% RSLogix 500 project Vacuum Feedback Control without PID.RSS, saved by version 8.30.00.16 %
PROJECT "UNTITLED"    % processor: Bul.1763 MicroLogix 1100 Series B %

PROGRAM FILES
  LAD 2   4 rungs
  LAD 3 "IO"  3 rungs
  LAD 4 "CTRL"  11 rungs

DATA FILES
  O0 OUTPUT  4 elements
  I1 INPUT  6 elements
  S2 STATUS  66 elements
  B3 BINARY  1 elements
  T4 TIMER  1 elements
  C5 COUNTER  1 elements
  R6 CONTROL  1 elements
  N7 INTEGER  7 elements
  F8 FLOAT  4 elements

LADDER 2
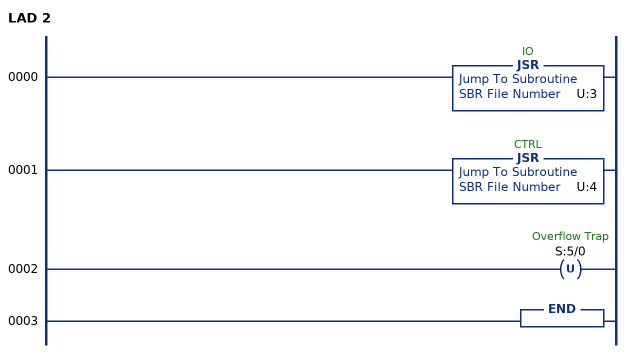
% Rung: 0 %
SOR JSR U:3 EOR
%   U:3  "IO" %
% Rung: 1 %
SOR JSR U:4 EOR
%   U:4  "CTRL" %
% Rung: 2 %
SOR OTU S:5/0 EOR
%   S:5/0  "Overflow Trap" %
% Rung: 3 %
SOR END EOR

LADDER 3 "IO"
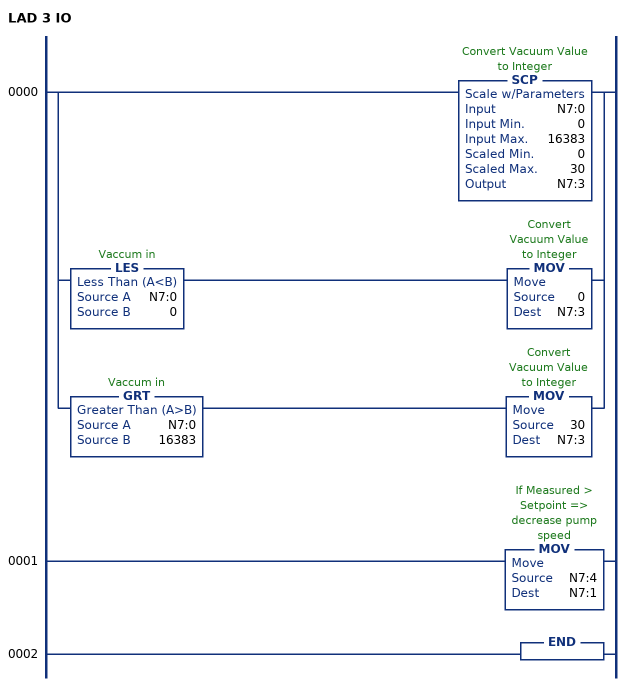
% Rung: 0 %
SOR BST SCP N7:0 0 16383 0 30 N7:3 NXB LES N7:0 0 MOV 0 N7:3 NXB GRT N7:0 16383 MOV 30 N7:3 BND EOR
%   N7:0  "Vaccum in" %
%   N7:3  "Convert Vacuum Value to Integer" %
% Rung: 1 %
SOR MOV N7:4 N7:1 EOR
%   N7:4  "(Measured - Setpoint)" %
%   N7:1  "If Measured > Setpoint => decrease pump speed" %
% Rung: 2 %
SOR END EOR

LADDER 4 "CTRL"
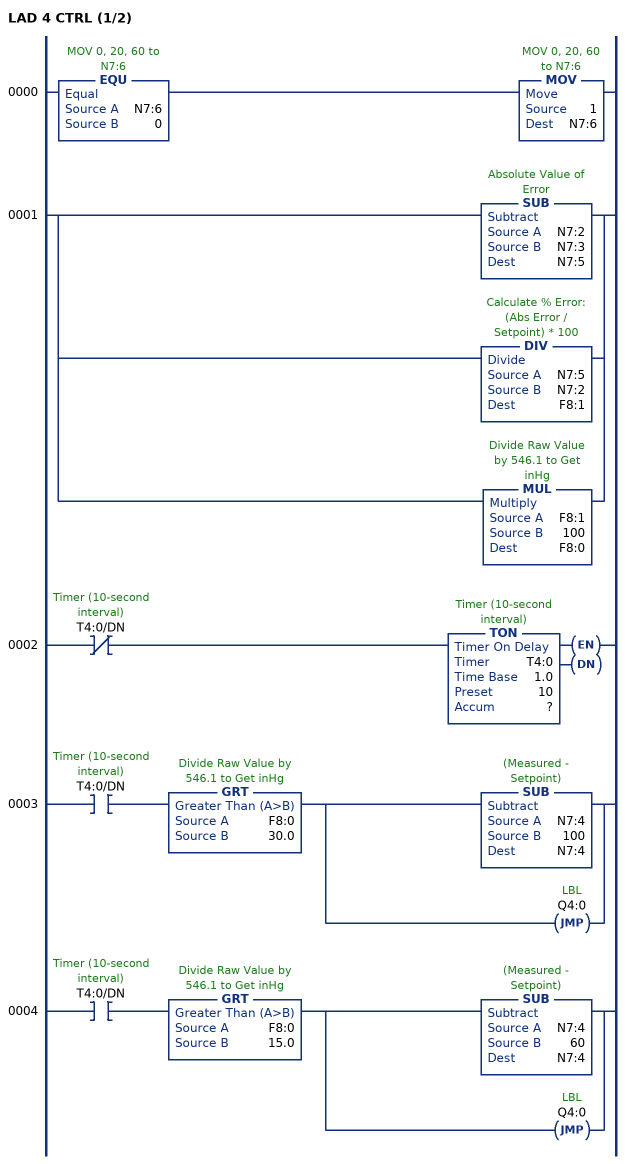
% Rung: 0 %
SOR EQU N7:6 0 MOV 1 N7:6 EOR
%   N7:6  "MOV 0, 20, 60 to N7:6" %
% Rung: 1 %
SOR BST SUB N7:2 N7:3 N7:5 NXB DIV N7:5 N7:2 F8:1 NXB MUL F8:1 100 F8:0 BND EOR
%   N7:2  "Calculate % Error: (Abs Error / Setpoint) * 100" %
%   N7:3  "Convert Vacuum Value to Integer" %
%   N7:5  "Absolute Value of Error" %
%   F8:1  "Calculate % Error: (Abs Error / Setpoint) * 100" %
%   F8:0  "Divide Raw Value by 546.1 to Get inHg" %
% Rung: 2 %  % edit flag set %
SOR XIO T4:0/DN TON T4:0 1.0 10 ? EOR
%   T4:0  "Timer (10-second interval)" %
% Rung: 3 %
SOR XIC T4:0/DN GRT F8:0 30.0 BST SUB N7:4 100 N7:4 NXB JMP Q4:0 BND EOR
%   T4:0  "Timer (10-second interval)" %
%   F8:0  "Divide Raw Value by 546.1 to Get inHg" %
%   N7:4  "(Measured - Setpoint)" %
%   Q4:0  "LBL" %
% Rung: 4 %
SOR XIC T4:0/DN GRT F8:0 15.0 BST SUB N7:4 60 N7:4 NXB JMP Q4:0 BND EOR
%   T4:0  "Timer (10-second interval)" %
%   F8:0  "Divide Raw Value by 546.1 to Get inHg" %
%   N7:4  "(Measured - Setpoint)" %
%   Q4:0  "LBL" %

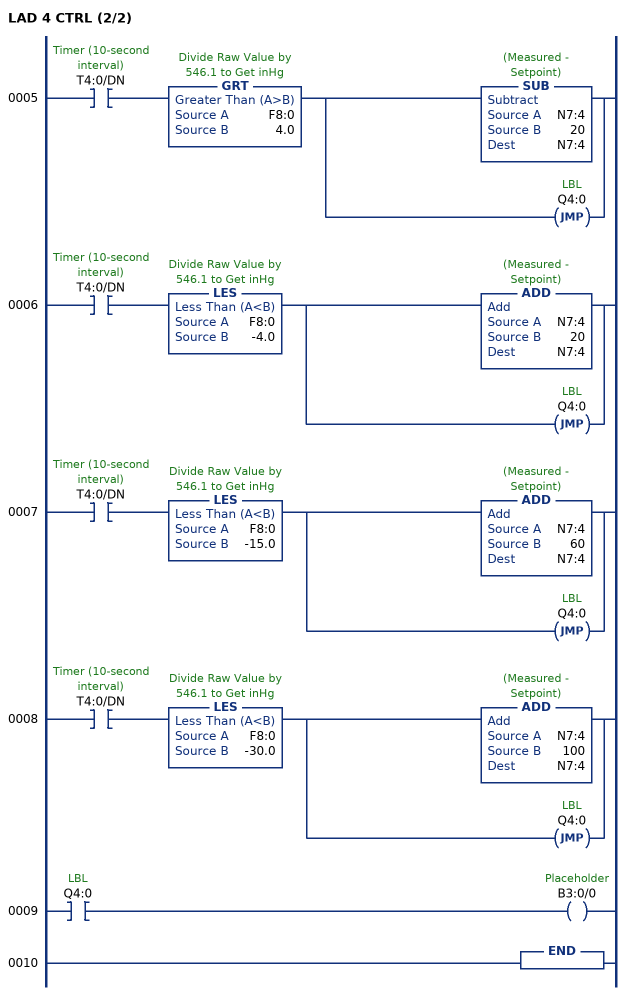
% Rung: 5 %
SOR XIC T4:0/DN GRT F8:0 4.0 BST SUB N7:4 20 N7:4 NXB JMP Q4:0 BND EOR
%   T4:0  "Timer (10-second interval)" %
%   F8:0  "Divide Raw Value by 546.1 to Get inHg" %
%   N7:4  "(Measured - Setpoint)" %
%   Q4:0  "LBL" %
% Rung: 6 %
SOR XIC T4:0/DN LES F8:0 -4.0 BST ADD N7:4 20 N7:4 NXB JMP Q4:0 BND EOR
%   T4:0  "Timer (10-second interval)" %
%   F8:0  "Divide Raw Value by 546.1 to Get inHg" %
%   N7:4  "(Measured - Setpoint)" %
%   Q4:0  "LBL" %
% Rung: 7 %
SOR XIC T4:0/DN LES F8:0 -15.0 BST ADD N7:4 60 N7:4 NXB JMP Q4:0 BND EOR
%   T4:0  "Timer (10-second interval)" %
%   F8:0  "Divide Raw Value by 546.1 to Get inHg" %
%   N7:4  "(Measured - Setpoint)" %
%   Q4:0  "LBL" %
% Rung: 8 %
SOR XIC T4:0/DN LES F8:0 -30.0 BST ADD N7:4 100 N7:4 NXB JMP Q4:0 BND EOR
%   T4:0  "Timer (10-second interval)" %
%   F8:0  "Divide Raw Value by 546.1 to Get inHg" %
%   N7:4  "(Measured - Setpoint)" %
%   Q4:0  "LBL" %
% Rung: 9 %  % edit flag set %
SOR XIC Q4:0 OTE B3:0/0 EOR
%   Q4:0  "LBL" %
%   B3:0/0  "Placeholder" %
% Rung: 10 %
SOR END EOR

OTHER DOCUMENTED ADDRESSES
  F8:2  "Raw Sensor Value to Floating Point Register"
  F8:3  "Convert Abs(Error) to Float"
